# EPICS substitutions: apps/svtCtrlApp/Db/svtR1-mpv-iseg.substitutions
# SVT HFCB HV & LV wiener modules substitution file
#  for iseg (HV) MX is slot # 1-10
file "db/iseg.db" {
pattern { HOST, HOSTNAME, MX }
  {"%(vmetlsvt1)","vmetlsvt1","7"}
  {"%(vmetlsvt1)","vmetlsvt1","8"}
}
#  for mpv (LV) MX is slot # 0-9
file "db/mpv.db" {
   pattern { HOST, HOSTNAME, MX }
  {"%(vmetlsvt1)","vmetlsvt1","0"}
  {"%(vmetlsvt1)","vmetlsvt1","1"}
  {"%(vmetlsvt1)","vmetlsvt1","2"}
  {"%(vmetlsvt1)","vmetlsvt1","3"}
  {"%(vmetlsvt1)","vmetlsvt1","4"}
}
